FUNCTION_BLOCK FB_Module_TEMPLATE EXTENDS FB_PMLModuleBase
VAR
    //Define the Sub modules here for this module. (If any)  Also set the Interfaces in the initialize method.
    (*fbSubModule1				: FB_ApplicationModule_TEMPLATE := (ModuleName :=  'Test Module 1');
	*)
    (*fbSubModule2				: FB_ApplicationModule_TEMPLATE := (ModuleName :=  'Test Module 2');
	*)
    //temporary array of module base interfaces to be copied over to the base class a_itfPackMLBase variable
    a_ITF_PackMLBase_init : ARRAY[1..MAX_NO_OF_SUBMODULES] OF ITF_PMLModuleBase
        := [ (*	fbSubModule1,
																							 	fbSubModule2*) ];

    //Define the components here for this module. (If any) Also set the Interfaces in the initialize method.
    (*fbComponent1				: FB_ComponentBase (Extension):= (Name := 'Test Component 1');
	*)
    (*fbComponent2				: FB_ComponentBase (Extension):= (Name := 'Test Component 2');
	*)
    //temporary array of module base interfaces to be copied over to the base class a_itfPackMLBase variable
    a_ITF_Components_init : ARRAY[1..GVL_PML_Base.MAX_NO_OF_COMPONENTS] OF ITF_ComponentBase := [ (*	fbComponent1,
																											fbComponent2*)
    ];

END_VAR

//*********************************************************
//Body of block is not called by base code, only implement application
//code in CyclicUpdate or in methods called by it or its subcalls
//*********************************************************

METHOD Aborted
CASE eMode OF
    //	====================================================================PRODUCTION MODE=========================================================	
    E_PMLUnitMode.ePMLUnitMode_Production:
        ;
    //	====================================================================MANUAL MODE=============================================================	
    E_PMLUnitMode.ePMLUnitMode_Manual:
        ;
    //	=====================================================================MAINTENANCE MODE=======================================================	
    E_PMLUnitMode.ePMLUnitMode_Maintenance:
        ;
    //	=====================================================================CUSTOM MODE 1==========================================================	
    (*	E_PMLUnitMode.ePMLUnitMode_YOURCUSTOMMODE		
		;*)
    //	======================================================================INVALID MODE==========================================================	
    E_PMLUnitMode.ePMLUnitMode_Invalid:
        ;
END_CASE
END_METHOD

METHOD Aborting
//bNoStateTasksToComplete := TRUE;		// Change to False if not used

//Implement state Tasks here
(*
IF (insert your completion conditions) THEN

bStateTasksComplete := TRUE;				//Once these actions are completed successfully, set bStateTasksComplete to allow the base code to advance once all children have also reached the proper state

END_IF
*)

SUPER^.Aborting();

(*	Reference State Machine for mode specific actions - Be sure to paste above the SUPER^ Call if used - Delete if not needed

CASE eMode OF
//	====================================================================PRODUCTION MODE=========================================================	
	E_PMLUnitMode.ePMLUnitMode_Production:			
		;
//	====================================================================MANUAL MODE=============================================================	
	E_PMLUnitMode.ePMLUnitMode_Manual:				
		;
//	=====================================================================MAINTENANCE MODE=======================================================	
	E_PMLUnitMode.ePMLUnitMode_Maintenance:			
		;	
//	=====================================================================CUSTOM MODE 1==========================================================	
(*	E_PMLUnitMode.ePMLUnitMode_YOURCUSTOMMODE		
		;*)
//	======================================================================INVALID MODE==========================================================	
	E_PMLUnitMode.ePMLUnitMode_Invalid:				
		;
END_CASE
*)
END_METHOD

METHOD Clearing
//bNoStateTasksToComplete := TRUE;		// Change to False if not used

//Implement state Tasks here
(*
IF (insert your completion conditions) THEN

bStateTasksComplete := TRUE;				//Once these actions are completed successfully, set bStateTasksComplete to allow the base code to advance once all children have also reached the proper state

END_IF
*)

SUPER^.Clearing();
(*	Reference State Machine for mode specific actions - Be sure to paste above the SUPER^ Call if used - Delete if not needed

CASE eMode OF
//	====================================================================PRODUCTION MODE=========================================================	
	E_PMLUnitMode.ePMLUnitMode_Production:			
		;
//	====================================================================MANUAL MODE=============================================================	
	E_PMLUnitMode.ePMLUnitMode_Manual:				
		;
//	=====================================================================MAINTENANCE MODE=======================================================	
	E_PMLUnitMode.ePMLUnitMode_Maintenance:			
		;	
//	=====================================================================CUSTOM MODE 1==========================================================	
(*	E_PMLUnitMode.ePMLUnitMode_YOURCUSTOMMODE		
		;*)
//	======================================================================INVALID MODE==========================================================	
	E_PMLUnitMode.ePMLUnitMode_Invalid:				
		;
END_CASE
*)
END_METHOD

METHOD Complete
CASE eMode OF
    //	====================================================================PRODUCTION MODE=========================================================	
    E_PMLUnitMode.ePMLUnitMode_Production:
        ;
    //	====================================================================MANUAL MODE=============================================================	
    E_PMLUnitMode.ePMLUnitMode_Manual:
        ;
    //	=====================================================================MAINTENANCE MODE=======================================================	
    E_PMLUnitMode.ePMLUnitMode_Maintenance:
        ;
    //	=====================================================================CUSTOM MODE 1==========================================================	
    (*	E_PMLUnitMode.ePMLUnitMode_YOURCUSTOMMODE		
		;*)
    //	======================================================================INVALID MODE==========================================================	
    E_PMLUnitMode.ePMLUnitMode_Invalid:
        ;
END_CASE
END_METHOD

METHOD Completing
//bNoStateTasksToComplete := TRUE;		// Change to False if not used

//Implement state Tasks here
(*
IF (insert your completion conditions) THEN

bStateTasksComplete := TRUE;				//Once these actions are completed successfully, set bStateTasksComplete to allow the base code to advance once all children have also reached the proper state

END_IF
*)

SUPER^.Completing();

(*	Reference State Machine for mode specific actions - Be sure to paste above the SUPER^ Call if used - Delete if not needed

CASE eMode OF
//	====================================================================PRODUCTION MODE=========================================================	
	E_PMLUnitMode.ePMLUnitMode_Production:			
		;
//	====================================================================MANUAL MODE=============================================================	
	E_PMLUnitMode.ePMLUnitMode_Manual:				
		;
//	=====================================================================MAINTENANCE MODE=======================================================	
	E_PMLUnitMode.ePMLUnitMode_Maintenance:			
		;	
//	=====================================================================CUSTOM MODE 1==========================================================	
(*	E_PMLUnitMode.ePMLUnitMode_YOURCUSTOMMODE		
		;*)
//	======================================================================INVALID MODE==========================================================	
	E_PMLUnitMode.ePMLUnitMode_Invalid:				
		;
END_CASE
*)
END_METHOD

// 
// Cyclic Code
METHOD CyclicLogic
VAR
    i : UDINT; //Generic iteration value
END_VAR
// Main loop of the parent module
SUPER^.CyclicLogic();
END_METHOD

METHOD Execute
CASE eMode OF
    //	====================================================================PRODUCTION MODE=========================================================	
    E_PMLUnitMode.ePMLUnitMode_Production:
        ;
    //	====================================================================MANUAL MODE=============================================================	
    E_PMLUnitMode.ePMLUnitMode_Manual:
        ;
    //	=====================================================================MAINTENANCE MODE=======================================================	
    E_PMLUnitMode.ePMLUnitMode_Maintenance:
        ;
    //	=====================================================================CUSTOM MODE 1==========================================================	
    (*	E_PMLUnitMode.ePMLUnitMode_YOURCUSTOMMODE		
		;*)
    //	======================================================================INVALID MODE==========================================================	
    E_PMLUnitMode.ePMLUnitMode_Invalid:
        ;
END_CASE
END_METHOD

METHOD Held
CASE eMode OF
    //	====================================================================PRODUCTION MODE=========================================================	
    E_PMLUnitMode.ePMLUnitMode_Production:
        ;
    //	====================================================================MANUAL MODE=============================================================	
    E_PMLUnitMode.ePMLUnitMode_Manual:
        ;
    //	=====================================================================MAINTENANCE MODE=======================================================	
    E_PMLUnitMode.ePMLUnitMode_Maintenance:
        ;
    //	=====================================================================CUSTOM MODE 1==========================================================	
    (*	E_PMLUnitMode.ePMLUnitMode_YOURCUSTOMMODE		
		;*)
    //	======================================================================INVALID MODE==========================================================	
    E_PMLUnitMode.ePMLUnitMode_Invalid:
        ;
END_CASE
END_METHOD

METHOD Holding
//bNoStateTasksToComplete := TRUE;		// Change to False if not used

//Implement state Tasks here
(*
IF (insert your completion conditions) THEN

bStateTasksComplete := TRUE;				//Once these actions are completed successfully, set bStateTasksComplete to allow the base code to advance once all children have also reached the proper state

END_IF
*)

SUPER^.Holding();

(*	Reference State Machine for mode specific actions - Be sure to paste above the SUPER^ Call if used - Delete if not needed

CASE eMode OF
//	====================================================================PRODUCTION MODE=========================================================	
	E_PMLUnitMode.ePMLUnitMode_Production:			
		;
//	====================================================================MANUAL MODE=============================================================	
	E_PMLUnitMode.ePMLUnitMode_Manual:				
		;
//	=====================================================================MAINTENANCE MODE=======================================================	
	E_PMLUnitMode.ePMLUnitMode_Maintenance:			
		;	
//	=====================================================================CUSTOM MODE 1==========================================================	
(*	E_PMLUnitMode.ePMLUnitMode_YOURCUSTOMMODE		
		;*)
//	======================================================================INVALID MODE==========================================================	
	E_PMLUnitMode.ePMLUnitMode_Invalid:				
		;
END_CASE
*)
END_METHOD

METHOD Idle
CASE eMode OF
    //	====================================================================PRODUCTION MODE=========================================================	
    E_PMLUnitMode.ePMLUnitMode_Production:
        ;
    //	====================================================================MANUAL MODE=============================================================	
    E_PMLUnitMode.ePMLUnitMode_Manual:
        ;
    //	=====================================================================MAINTENANCE MODE=======================================================	
    E_PMLUnitMode.ePMLUnitMode_Maintenance:
        ;
    //	=====================================================================CUSTOM MODE 1==========================================================	
    (*	E_PMLUnitMode.ePMLUnitMode_YOURCUSTOMMODE		
		;*)
    //	======================================================================INVALID MODE==========================================================	
    E_PMLUnitMode.ePMLUnitMode_Invalid:
        ;
END_CASE
END_METHOD

METHOD Initialize
VAR
    i : UDINT; //Generic iteration value
END_VAR
// Define the interfaces to the different subunits (Must take place before SUPER^.initialize call)
FOR i := 1 TO MAX_NO_OF_SUBMODULES DO
    a_ITF_PackMLBase[i] := a_ITF_PackMLBase_init[i];
END_FOR

FOR i := 1 TO MAX_NO_OF_COMPONENTS DO
    a_ITF_Components[i] := a_ITF_Components_init[i];
END_FOR

// Init of the parent class object (Must be called AFTER most local init code, since the sub module interface array assignments should be made here, and then operated on within the module base init
SUPER^.Initialize();
END_METHOD

METHOD Resetting
//bNoStateTasksToComplete := TRUE;		// Change to False if not used

//Implement state Tasks here
(*
IF (insert your completion conditions) THEN

bStateTasksComplete := TRUE;				//Once these actions are completed successfully, set bStateTasksComplete to allow the base code to advance once all children have also reached the proper state

END_IF
*)

SUPER^.Resetting();

(*	Reference State Machine for mode specific actions - Be sure to paste above the SUPER^ Call if used - Delete if not needed

CASE eMode OF
//	====================================================================PRODUCTION MODE=========================================================	
	E_PMLUnitMode.ePMLUnitMode_Production:			
		;
//	====================================================================MANUAL MODE=============================================================	
	E_PMLUnitMode.ePMLUnitMode_Manual:				
		;
//	=====================================================================MAINTENANCE MODE=======================================================	
	E_PMLUnitMode.ePMLUnitMode_Maintenance:			
		;	
//	=====================================================================CUSTOM MODE 1==========================================================	
(*	E_PMLUnitMode.ePMLUnitMode_YOURCUSTOMMODE		
		;*)
//	======================================================================INVALID MODE==========================================================	
	E_PMLUnitMode.ePMLUnitMode_Invalid:				
		;
END_CASE
*)
END_METHOD

METHOD Starting
//bNoStateTasksToComplete := TRUE;		// Change to False if not used

//Implement state Tasks here
(*
IF (insert your completion conditions) THEN

bStateTasksComplete := TRUE;				//Once these actions are completed successfully, set bStateTasksComplete to allow the base code to advance once all children have also reached the proper state

END_IF
*)

SUPER^.Starting();

(*	Reference State Machine for mode specific actions - Be sure to paste above the SUPER^ Call if used - Delete if not needed

CASE eMode OF
//	====================================================================PRODUCTION MODE=========================================================	
	E_PMLUnitMode.ePMLUnitMode_Production:			
		;
//	====================================================================MANUAL MODE=============================================================	
	E_PMLUnitMode.ePMLUnitMode_Manual:				
		;
//	=====================================================================MAINTENANCE MODE=======================================================	
	E_PMLUnitMode.ePMLUnitMode_Maintenance:			
		;	
//	=====================================================================CUSTOM MODE 1==========================================================	
(*	E_PMLUnitMode.ePMLUnitMode_YOURCUSTOMMODE		
		;*)
//	======================================================================INVALID MODE==========================================================	
	E_PMLUnitMode.ePMLUnitMode_Invalid:				
		;
END_CASE
*)
END_METHOD

METHOD Stopped
CASE eMode OF
    //	====================================================================PRODUCTION MODE=========================================================	
    E_PMLUnitMode.ePMLUnitMode_Production:
        ;
    //	====================================================================MANUAL MODE=============================================================	
    E_PMLUnitMode.ePMLUnitMode_Manual:
        ;
    //	=====================================================================MAINTENANCE MODE=======================================================	
    E_PMLUnitMode.ePMLUnitMode_Maintenance:
        ;
    //	=====================================================================CUSTOM MODE 1==========================================================	
    (*	E_PMLUnitMode.ePMLUnitMode_YOURCUSTOMMODE		
		;*)
    //	======================================================================INVALID MODE==========================================================	
    E_PMLUnitMode.ePMLUnitMode_Invalid:
        ;
END_CASE
END_METHOD

METHOD Stopping
//bNoStateTasksToComplete := TRUE;		// Change to False if not used

//Implement state Tasks here
(*
IF (insert your completion conditions) THEN

bStateTasksComplete := TRUE;				//Once these actions are completed successfully, set bStateTasksComplete to allow the base code to advance once all children have also reached the proper state

END_IF
*)

SUPER^.Stopping();

(*	Reference State Machine for mode specific actions - Be sure to paste above the SUPER^ Call if used - Delete if not needed

CASE eMode OF
//	====================================================================PRODUCTION MODE=========================================================	
	E_PMLUnitMode.ePMLUnitMode_Production:			
		;
//	====================================================================MANUAL MODE=============================================================	
	E_PMLUnitMode.ePMLUnitMode_Manual:				
		;
//	=====================================================================MAINTENANCE MODE=======================================================	
	E_PMLUnitMode.ePMLUnitMode_Maintenance:			
		;	
//	=====================================================================CUSTOM MODE 1==========================================================	
(*	E_PMLUnitMode.ePMLUnitMode_YOURCUSTOMMODE		
		;*)
//	======================================================================INVALID MODE==========================================================	
	E_PMLUnitMode.ePMLUnitMode_Invalid:				
		;
END_CASE
*)
END_METHOD

METHOD Suspended
CASE eMode OF
    //	====================================================================PRODUCTION MODE=========================================================	
    E_PMLUnitMode.ePMLUnitMode_Production:
        ;
    //	====================================================================MANUAL MODE=============================================================	
    E_PMLUnitMode.ePMLUnitMode_Manual:
        ;
    //	=====================================================================MAINTENANCE MODE=======================================================	
    E_PMLUnitMode.ePMLUnitMode_Maintenance:
        ;
    //	=====================================================================CUSTOM MODE 1==========================================================	
    (*	E_PMLUnitMode.ePMLUnitMode_YOURCUSTOMMODE		
		;*)
    //	======================================================================INVALID MODE==========================================================	
    E_PMLUnitMode.ePMLUnitMode_Invalid:
        ;
END_CASE
END_METHOD

METHOD Suspending
//bNoStateTasksToComplete := TRUE;		// Change to False if not used

//Implement state Tasks here
(*
IF (insert your completion conditions) THEN

bStateTasksComplete := TRUE;				//Once these actions are completed successfully, set bStateTasksComplete to allow the base code to advance once all children have also reached the proper state

END_IF
*)

SUPER^.Suspending();

(*	Reference State Machine for mode specific actions - Be sure to paste above the SUPER^ Call if used - Delete if not needed

CASE eMode OF
//	====================================================================PRODUCTION MODE=========================================================	
	E_PMLUnitMode.ePMLUnitMode_Production:			
		;
//	====================================================================MANUAL MODE=============================================================	
	E_PMLUnitMode.ePMLUnitMode_Manual:				
		;
//	=====================================================================MAINTENANCE MODE=======================================================	
	E_PMLUnitMode.ePMLUnitMode_Maintenance:			
		;	
//	=====================================================================CUSTOM MODE 1==========================================================	
(*	E_PMLUnitMode.ePMLUnitMode_YOURCUSTOMMODE		
		;*)
//	======================================================================INVALID MODE==========================================================	
	E_PMLUnitMode.ePMLUnitMode_Invalid:				
		;
END_CASE
*)
END_METHOD

METHOD Undefined
CASE eMode OF
    //	====================================================================PRODUCTION MODE=========================================================	
    E_PMLUnitMode.ePMLUnitMode_Production:
        ;
    //	====================================================================MANUAL MODE=============================================================	
    E_PMLUnitMode.ePMLUnitMode_Manual:
        ;
    //	=====================================================================MAINTENANCE MODE=======================================================	
    E_PMLUnitMode.ePMLUnitMode_Maintenance:
        ;
    //	=====================================================================CUSTOM MODE 1==========================================================	
    (*	E_PMLUnitMode.ePMLUnitMode_YOURCUSTOMMODE		
		;*)
    //	======================================================================INVALID MODE==========================================================	
    E_PMLUnitMode.ePMLUnitMode_Invalid:
        ;
END_CASE
END_METHOD

METHOD Unholding
//bNoStateTasksToComplete := TRUE;		// Change to False if not used

//Implement state Tasks here
(*
IF (insert your completion conditions) THEN

bStateTasksComplete := TRUE;				//Once these actions are completed successfully, set bStateTasksComplete to allow the base code to advance once all children have also reached the proper state

END_IF
*)

SUPER^.Unholding();

(*	Reference State Machine for mode specific actions - Be sure to paste above the SUPER^ Call if used - Delete if not needed

CASE eMode OF
//	====================================================================PRODUCTION MODE=========================================================	
	E_PMLUnitMode.ePMLUnitMode_Production:			
		;
//	====================================================================MANUAL MODE=============================================================	
	E_PMLUnitMode.ePMLUnitMode_Manual:				
		;
//	=====================================================================MAINTENANCE MODE=======================================================	
	E_PMLUnitMode.ePMLUnitMode_Maintenance:			
		;	
//	=====================================================================CUSTOM MODE 1==========================================================	
(*	E_PMLUnitMode.ePMLUnitMode_YOURCUSTOMMODE		
		;*)
//	======================================================================INVALID MODE==========================================================	
	E_PMLUnitMode.ePMLUnitMode_Invalid:				
		;
END_CASE
*)
END_METHOD

METHOD Unsuspending
//bNoStateTasksToComplete := TRUE;		// Change to False if not used

//Implement state Tasks here
(*
IF (insert your completion conditions) THEN

bStateTasksComplete := TRUE;				//Once these actions are completed successfully, set bStateTasksComplete to allow the base code to advance once all children have also reached the proper state

END_IF
*)

SUPER^.Unsuspending();

(*	Reference State Machine for mode specific actions - Be sure to paste above the SUPER^ Call if used - Delete if not needed

CASE eMode OF
//	====================================================================PRODUCTION MODE=========================================================	
	E_PMLUnitMode.ePMLUnitMode_Production:			
		;
//	====================================================================MANUAL MODE=============================================================	
	E_PMLUnitMode.ePMLUnitMode_Manual:				
		;
//	=====================================================================MAINTENANCE MODE=======================================================	
	E_PMLUnitMode.ePMLUnitMode_Maintenance:			
		;	
//	=====================================================================CUSTOM MODE 1==========================================================	
(*	E_PMLUnitMode.ePMLUnitMode_YOURCUSTOMMODE		
		;*)
//	======================================================================INVALID MODE==========================================================	
	E_PMLUnitMode.ePMLUnitMode_Invalid:				
		;
END_CASE
*)
END_METHOD

END_FUNCTION_BLOCK

(* stored: Version 1.1.0.1, ProductVersion 3.1.4024.11
   POU FB_Module_TEMPLATE: Id {44c00981-3585-4538-bbce-d21beee256d9}, SpecialFunc None
   Folder 01_SUPER_Overrides: Id {f8d8b220-72f9-48a9-9ea0-e208740f789c}
   Folder 01_Properties: Id {057d9d1a-ee49-4f19-8a8e-42e6aa4c339e}
   Folder 01_Config: Id {331100b9-f98f-4747-8f54-d0fce7db7a42}
   Folder 02_Control: Id {ae3e5afd-d53d-4093-8ebe-aff2e7e7d938}
   Folder 03_Status: Id {33277d99-4da9-43f5-93be-20a601b15ef0}
   Folder 02_Methods: Id {19c5cdd7-570a-4a8c-8c2e-0d3729a276d3}
   Folder 03_TransitionStates: Id {dc4f9408-7e17-43e6-92f9-f3fb8ef0556c}
   Folder 04_PrimaryStates: Id {38edaf77-9798-4b46-b36f-091ed1d56038}
   Folder 02_Properties: Id {622b930f-94e4-47af-8e64-1bce8c192706}
   Folder 01_Config: Id {60f94e06-65b6-4e11-88a4-cbfadd90a020}
   Folder 02_Control: Id {0df8385a-1171-4989-abde-723998077e92}
   Folder 03_Status: Id {49d473b9-52dd-4d23-948d-b6a2dc357f76}
   Folder 03_Methods: Id {7a7ecdb0-5f2b-448e-937a-8df184a6286e}
   Method Aborted: Id {115f0d92-9b74-4207-98d9-01bbe419601d}
   Method Aborting: Id {f8525f20-f595-4df6-a37f-5015b53b7fec}
   Method Clearing: Id {ff990ee6-ab5b-4b58-a115-900e05af0a3f}
   Method Complete: Id {b03e4f78-5c1e-4da5-bdad-0d056e0792b4}
   Method Completing: Id {b10641f1-5701-4ac0-9217-732c3b77e29d}
   Method CyclicLogic: Id {12422e5e-a5c0-4929-9ad9-b99a74293d93}
   Method Execute: Id {4241bd48-fc56-47ed-a03f-f06bee0b8de4}
   Method Held: Id {8b7d10d4-56d1-44a0-b483-b75edbbd5aa4}
   Method Holding: Id {13997f8d-82e7-42dd-a219-e0992db665ee}
   Method Idle: Id {ba890787-538d-464f-9cf3-cf1fe940fbce}
   Method Initialize: Id {442f3bf5-5552-4c37-b5b2-a49ca36d752d}
   Method Resetting: Id {7565530e-bb29-4323-9478-8b5cf80eeec5}
   Method Starting: Id {d7fb0679-54a8-4166-bc3f-65cfbf96a41a}
   Method Stopped: Id {98c12991-c1d2-4cb1-a15e-a79edff2bbe1}
   Method Stopping: Id {a2353e86-b48b-4844-8cfa-38fb6356963a}
   Method Suspended: Id {abaf0f7b-1797-42dc-8264-67066b23666c}
   Method Suspending: Id {4a96f516-2ab2-4259-856f-ce4b47b47f7d}
   Method Undefined: Id {3c51e684-53f6-47f3-bf4c-ce7a21a58158}
   Method Unholding: Id {3c1714cd-0eb3-473b-b55c-c60b1d11d33e}
   Method Unsuspending: Id {922b0ce4-9914-4a7f-862d-70e53c049c14} *)
